PROGRAM F_TERMOREG
VAR_INPUT
	Func:e_funcio;
END_VAR
VAR
	///Activa
	xActv: BOOL;
	///Parametros
	wP_TempFinal: WORD;
	wP_Mant: WORD;
	wP_Grad: WORD;
	xP_Pasajes: BOOL;
	///Fin Funcion
	xFiFunc: BOOL;
	
	xIniciaTermo: BOOL;
	tDelayinicio: Ton;
	rUltimaTermp: REAL;
	iTiempoPaso: INT;
	rTempFinal: REAL;
	iMant: INT;
	rGrad: REAL;
	xPasajes: BOOL;
	xPulseReg: BOOL;
	Cont: ctu;
	manrs: BOOL;
	wcanttt: WORD;
	rGradProg: REAL;
	tDelayPumpOK: Ton;
	xPumpRuns: BOOL;
	xGrad0: BOOL;
	xSegOk: BOOL;
	xStopSP: BOOL;
	x: INT;
	Termo: fBTermo;
	xPauseMant: BOOL;
	tTmpMant: TMP_P;
	xNoMant: BOOL;
	iTmpMant: INT;
	tFinSinMant: Ton;
	tTiempoIgualacion: TIME := TIME#15s0ms;
	xFiT_NoMant: BOOL;
	tFinConMant: Ton;
	FinFuncion: BOOL;
	Z_xVapor: BOOL;
	z_xEnfria: BOOL;
	z_rApertVapor: REAL;
	z_rApertEnfria: REAL;
	z_xRetonoCond: BOOL;
	rI_PID: LREAL;
	dwTempsMsnt: DINT;
	xTempMinima: BOOL;
	xABombaCircParada: BOOL;
END_VAR

//carga valores funcion

xActv:= Func.Actv_Funcio;

rTempFinal:=	WORD_TO_REAL(func.ParamFunc[1]);
rGrad:=			WORD_TO_REAL(func.ParamFunc[2]);
iMant:=			WORD_TO_INT(func.ParamFunc[3]);
xPasajes:= 		(func.ParamFunc[2]>0);	
 

//Inicia Termo
tDelayinicio(IN:= 	xActv AND 					//Funcion activa
				 	NOT(ATL.PE_COM.xResetFunc) , 	//No hay reset de tiempo funcion
				PT:= T#1S);
xIniciaTermo:= 	tDelayinicio.Q ;

//MEMORIZAR DATOS
//Memorizar Tiempo de paso
//IF xFuncActv AND NOT(xIniciaTermo) THEN
//	iTiempoPaso:=_00_Winch.TempsAnt1[1];
//END_IF

//Calculo Gradiente
IF rGrad=0
	THEN
	rGradProg := Mc._02_TEMP.iPFDefauldGrad;
	xGrad0:=TRUE;
	ELSIF   xPasajes>0
		THEN
		xGrad0:=FALSE;
		//Calcular Gradiente por pasajes
		//Si el tiempo de paso es cero se carga 60seg	
		IF iTiempoPaso=0 THEN		
			iTiempoPaso:=60;
		END_IF	
		rGradProg:= (rGrad*60.0)/INT_TO_REAL(iTiempoPaso);					
		ELSE
		xGrad0:=FALSE;
		rGradProg:=rGrad;	
END_IF


//Tiempo de Bomba en marcha para iniciar Termo
tDelayPumpOK(IN:= Mc._09_CPUMP.b450_CircPump.xOK , PT:= INT_TO_TIME(MC._02_TEMP.iPFTimeOfPumpToRun)*1000 );
xPumpRuns:=tDelayPumpOK.Q;

//Seguridades Para Termo	
xSegOk:=	Mc._06_LEVEL.xLvl_min AND 			//Nivel minimo
			NOT(Mc._01_SEG.xMcOpen) AND 		//Maquina Oberta
			NOT(Mc._01_SEG.xMaxPresTemp) AND	//No hi ha ni max temp ni max Press
			Mc._09_CPUMP.b450_CircPump.xOK	AND		//Bomba girando
			xPumpRuns AND					//Bomba esta en marcha por un tiempo determinado
			NOT(Mc._02_temp.xPT100Failure)  ;	//Fallo PT-100
			//FALTA DIF >5ºC

//parar la consigna
xStopSP:= 	NOT(xSegOK) AND 
			NOT(xPumpRuns);				 
			//Falta maquina pausada

//------------------------------------------------------------------------

Termo(
	TermoActv:= 			xIniciaTermo, //AND xPumpRuns, 
	TemperaturaReal:= 		Mc._02_TEMP.rMacTemperature, 
	TemperaturaFinal:=		rTempFinal, 
	Gradient:= 				rGradProg, 
	t_Manteniment:= 		iMant, 
	Pols:= 					_00_Generales.Pulso_1s.xFlanco, 
	PausaExterior:= 		xStopSP OR NOT xPumpRuns, 
	GrausPerIntegracio:= 	Mc._02_TEMP.iPFGradIntegra, 
	GrausForzarCal:= 		Mc._02_TEMP.iPFGradForzCal, 
	ReIniciarTermo:= 		FALSE, 
	TmoSegConmutacion:= 	INT_TO_DWORD(Mc._02_TEMP.iPFTmpComutac), 
	ConmutacioEnManteniment:= Mc._02_TEMP.iPFGradComutac, 
	BandaProporcional:= 	Mc._02_TEMP.iPFPID_P, 
	PartIntergral:= 		Mc._02_TEMP.iPFPID_I, 
	PartDerivada:= 			Mc._02_TEMP.iPFPID_D, 
	T_periode:= 			0.01, 
	SeguretatOK:= 			xSegOk, 
	ObrirPurgaenRepos:= 	FALSE, 
	t_Purga:= 				0, 
	TemperaturaPerInici:= 	Mc._02_TEMP.rMacTemperature, 
	NO_Reset:= 				FALSE, 
	
	 );

Mc._02_TEMP.rTempImp:= F_TERMOREG.Termo.TemperaturaImposada;
//Control MAnteniment-------------------------------------------
//Pausa¡ Manteniment
xPauseMant:=	NOT(Mc._09_CPUMP.b450_CircPump.xOK) OR
				MC._00_GENERAL.xMcPaused;
//Calculo Tiempo Mantenimiento por pasaje

IF iMant=0
	THEN
	xNoMant:=TRUE;
	ELSIF xPasajes
		THEN
		xNoMant:=FALSE;
		iTmpMant:= iMant*iTiempoPaso;
		ELSE
		xNoMant:=FALSE;
		iTmpMant:= iMant;		
END_IF

				
//Tiempo Mantenimiento
tTmpMant(
	xIN:= 		Termo.EnManteniment, 
	xPausa:= 	xPauseMant, 
	dwSegons:= 	INT_TO_DWORD(iTmpMant)*60, 
	 );
dwTempsMsnt:= (iMant*60)-(REAL_TO_INT(tTmpMant.rTsegons));


//FinFuncion --------------------------------------
//Sin Mantenimiento tiempo de igualar temperatura
tFinSinMant(	IN:= Termo.EnManteniment, 
				PT:=tTiempoIgualacion  );
xFiT_NoMant:= tFinSinMant.Q AND xNoMant;
//Con mantenimiento
tFinConMant(IN:=tTmpMant.xQ , 
			PT:= T#5S );
//Enfriar a temperartura baja			
xTempMinima:= termo.AiguaRefredament AND ( rTempFinal< Mc._02_TEMP.iPFTempMinCool);


			
//Finalizar
FinFuncion:=xFiT_NoMant OR tFinConMant.Q OR xTempMinima;
xFiFunc:=FinFuncion;

//======================================================================================
// Alarmas
//======================================================================================
xABombaCircParada:= xActv AND NOT (Mc._09_CPUMP.b450_CircPump.xOK);

//=========================================================================================================
// Activar salidas
//=========================================================================================================

Z_xVapor:= 		Termo.Vapor;
z_xEnfria:= 	Termo.AiguaRefredament;
z_rApertVapor:=	Termo.Apertura_Vapor;
z_rApertEnfria:=Termo.Apertura_Refreda;

//Retorn condensados
z_xRetonoCond:= z_xVapor AND (*Mc.TEMP.xRetCond AND*) F_TERMOREG.Termo.Actv_RetornVapor ;

END_PROGRAM

(* stored: Version 1.1.0.1, ProductVersion 3.1.4024.10
   POU F_TERMOREG: Id {aff765c8-6a0e-44f4-85fb-ca7fda0e5db0}, SpecialFunc None *)
